// Mitsubishi GX Works2 project: BookEX6_10 String   PLC: Q13UDV

// global labels: Global
VAR_GLOBAL
  bVar0 AT M5000 : BOOL;
  abArray0 AT M5010 : ARRAY [0..49] OF BOOL;
  sStr0 AT D5000 : STRING[199];
  sStr1 AT D5100 : STRING[199];
  sStr2 AT D5200 : STRING[199];
  sStr3 AT D5300 : STRING[199];
  sStr4 AT D5400 : STRING[199];
  sStr5 AT D5500 : STRING[199];
  sStr6 AT D5600 : STRING[199];
  sStr7 AT D5700 : STRING[199];
  sStr8 AT D5800 : STRING[199];
  sStr9 AT D5900 : STRING[199];
  iVar0 AT D4500 : INT;
  iVar1 AT D4501 : INT;
  iVar2 AT D4502 : INT;
  iVar3 AT D4503 : INT;
  iVar4 AT D4504 : INT;
  iVar5 AT D4505 : INT;
  iVar6 AT D4506 : INT;
  iVar7 AT D4507 : INT;
  iVar8 AT D4508 : INT;
  iVar9 AT D4509 : INT;
  dVar0 AT D4510 : DINT;
  dVar1 AT D4512 : DINT;
  dVar2 AT D4514 : DINT;
  dVar3 AT D4516 : DINT;
  dVar4 AT D4518 : DINT;
  dVar5 AT D4520 : DINT;
  dVar6 AT D4522 : DINT;
  dVar7 AT D4524 : DINT;
  dVar8 AT D4526 : DINT;
  dVar9 AT D4528 : DINT;
  wVar0 AT D4530 : WORD;
  wVar1 AT D4531 : WORD;
  wVar2 AT D4532 : WORD;
  wVar3 AT D4533 : WORD;
  wVar4 AT D4534 : WORD;
  wVar5 AT D4535 : WORD;
  wVar6 AT D4536 : WORD;
  wVar7 AT D4537 : WORD;
  wVar8 AT D4538 : WORD;
  wVar9 AT D4539 : WORD;
  dwVar0 AT D4540 : DWORD;
  dwVar1 AT D4542 : DWORD;
  dwVar2 AT D4544 : DWORD;
  dwVar3 AT D4546 : DWORD;
  dwVar4 AT D4548 : DWORD;
  dwVar5 AT D4550 : DWORD;
  dwVar6 AT D4552 : DWORD;
  dwVar7 AT D4554 : DWORD;
  dwVar8 AT D4556 : DWORD;
  dwVar9 AT D4558 : DWORD;
  fsVar0 AT D4560 : REAL;
  fsVar1 AT D4562 : REAL;
  fsVar2 AT D4564 : REAL;
  fsVar3 AT D4566 : REAL;
  fsVar4 AT D4568 : REAL;
  fsVar5 AT D4570 : REAL;
  fsVar6 AT D4572 : REAL;
  fsVar7 AT D4574 : REAL;
  fsVar8 AT D4576 : REAL;
  fsVar9 AT D4578 : REAL;
  fdVar0 AT D4580 : LREAL;
  tTime0 AT D4620 : TIME;
  tTime1 AT D4622 : TIME;
  tTime2 AT D4624 : TIME;
  tTime3 AT D4626 : TIME;
  tTime4 AT D4628 : TIME;
  tTime5 AT D4630 : TIME;
  tTime6 AT D4632 : TIME;
  tTime7 AT D4634 : TIME;
  tTime8 AT D4636 : TIME;
  tTime9 AT D4638 : TIME;
  tTime10 AT D4640 : TIME;
  bVar1 AT M5001 : BOOL;
  bVar2 AT M5002 : BOOL;
  bVar3 AT M5003 : BOOL;
  bVar4 AT M5004 : BOOL;
  bVar5 AT M5005 : BOOL;
  bVar6 AT M5006 : BOOL;
  bVar7 AT M5007 : BOOL;
  bVar8 AT M5008 : BOOL;
  bVar9 AT M5009 : BOOL;
  abArray1 AT M5060 : ARRAY [0..49] OF BOOL;
  abArray2 AT M5110 : ARRAY [0..49] OF BOOL;
  abArray3 AT M5160 : ARRAY [0..49] OF BOOL;
  abArray4 AT M5210 : ARRAY [0..49] OF BOOL;
  abArray5 AT M5260 : ARRAY [0..49] OF BOOL;
  abArray6 AT M5310 : ARRAY [0..49] OF BOOL;
  abArray7 AT M5360 : ARRAY [0..49] OF BOOL;
  abArray8 AT M5410 : ARRAY [0..49] OF BOOL;
  abArray9 AT M5460 : ARRAY [0..49] OF BOOL;
  fdVar1 AT D4584 : LREAL;
  fdVar2 AT D4588 : LREAL;
  fdVar3 AT D4592 : LREAL;
  fdVar4 AT D4596 : LREAL;
  fdVar5 AT D4600 : LREAL;
  fdVar6 AT D4604 : LREAL;
  fdVar7 AT D4608 : LREAL;
  fdVar8 AT D4612 : LREAL;
  fdVar9 AT D4616 : LREAL;
END_VAR
// user libraries (not included): HMI

FUNCTION ChkALNUM
VAR_INPUT
  s_IN : STRING[199];
END_VAR
VAR
  ix : INT;
  iLeng : INT;
  iChar : INT;
  sTmpStr : STRING[199];
END_VAR
;
sTmpStr := s_IN;
LEN_E(TRUE, s_IN, iLeng);
IF iLeng = 0 THEN
	ChkALNUM := FALSE;
	RETURN;
END_IF;
FOR ix := 1 TO iLeng DO
	iChar := GET_INT_ADDR(sTmpStr) MOD 256;
	IF NOT ((iChar > H2F AND iChar < H3A) OR (iChar > H40 AND iChar < H5B) OR (iChar > H60 AND iChar < H7B)) THEN
		ChkALNUM := FALSE;
		RETURN;
	END_IF;
	sTmpStr := DELETE(sTmpStr, 1, 1);
END_FOR;
ChkALNUM := TRUE;
END_FUNCTION

FUNCTION ChkALPHA
VAR_INPUT
  s_IN : STRING[199];
END_VAR
VAR
  ix : INT;
  iLeng : INT;
  iChar : INT;
  sTmpStr : STRING[199];
END_VAR
;
sTmpStr := s_IN;
LEN_E(TRUE, s_IN, iLeng);
IF iLeng = 0 THEN
	ChkALPHA := FALSE;
	RETURN;
END_IF;
FOR ix := 1 TO iLeng DO
	iChar := GET_INT_ADDR(sTmpStr) MOD 256;
	IF NOT ((iChar > H40 AND iChar < H5B) OR (iChar > H60 AND iChar < H7B)) THEN
		ChkALPHA := FALSE;
		RETURN;
	END_IF;
	sTmpStr := DELETE(sTmpStr, 1, 1);
END_FOR;
ChkALPHA := TRUE;
END_FUNCTION

FUNCTION ChkHEXSTR
VAR_INPUT
  s_IN : STRING[199];
END_VAR
VAR
  ix : INT;
  iLeng : INT;
  iChar : INT;
  sTmpStr : STRING[199];
END_VAR
;
sTmpStr := s_IN;
LEN_E(TRUE, s_IN, iLeng);
IF iLeng = 0 THEN
	ChkHEXSTR := FALSE;
	RETURN;
END_IF;
FOR ix := 1 TO iLeng DO
	iChar := GET_INT_ADDR(sTmpStr) MOD 256;
	IF NOT ((iChar > H2F AND iChar < H3A) OR (iChar > H40 AND iChar < H47) OR (iChar > H60 AND iChar < H67)) THEN
		ChkHEXSTR := FALSE;
		RETURN;
	END_IF;
	sTmpStr := DELETE(sTmpStr, 1, 1);
END_FOR;
ChkHEXSTR := TRUE;
END_FUNCTION

FUNCTION ChkNUM
VAR_INPUT
  s_IN : STRING[199];
END_VAR
VAR
  ix : INT;
  iLeng : INT;
  iChar : INT;
  sTmpStr : STRING[199];
END_VAR
;
sTmpStr := s_IN;
LEN_E(TRUE, s_IN, iLeng);
IF iLeng = 0 THEN
	ChkNUM := FALSE;
	RETURN;
END_IF;
FOR ix := 1 TO iLeng DO
	iChar := GET_INT_ADDR(sTmpStr) MOD 256;
	IF NOT (iChar > H2F AND iChar < H3A) THEN
		ChkNUM := FALSE;
		RETURN;
	END_IF;
	sTmpStr := DELETE(sTmpStr, 1, 1);
END_FOR;
ChkNUM := TRUE;
END_FUNCTION

FUNCTION FindNUM
VAR_INPUT
  s_IN : STRING[199];
END_VAR
VAR
  ix : INT;
  iLeng : INT;
  iChar : INT;
  sTmpStr : STRING[199];
END_VAR
VAR_INPUT
  b_Num : BOOL;
END_VAR
;
sTmpStr := s_IN;
LEN_E(TRUE, s_IN, iLeng);
IF iLeng = 0 THEN
	FindNUM := 0;
	RETURN;
END_IF;
FOR ix := 1 TO iLeng DO
	iChar := GET_INT_ADDR(sTmpStr) MOD 256;
	IF (b_Num AND (iChar > H2F AND iChar < H3A)) OR 
		(NOT b_Num AND  NOT (iChar > H2F AND iChar < H3A)) THEN
		FindNUM := ix;
		RETURN;
	END_IF;
	sTmpStr := DELETE(sTmpStr, 1, 1);
END_FOR;
FindNUM := 0;
END_FUNCTION

FUNCTION MirrorStr
VAR_INPUT
  s_IN : STRING[199];
END_VAR
VAR
  ix : INT;
  iLeng : INT;
  sChar : STRING[1];
  sTmpStr : STRING[199];
  sTmpStr2 : STRING[199];
  sTmpStr1 : STRING[199];
END_VAR
;
sTmpStr := s_IN;
LEN_E(TRUE, s_IN, iLeng);
IF iLeng < 2 THEN
	MirrorStr := sTmpStr;
	RETURN;
END_IF;
sTmpStr2 := '';
FOR ix := iLeng TO 1 BY -1 DO 
	RIGHT_E(TRUE, sTmpStr, 1, sChar);
(*	STRDEL(TRUE, ix, 1, sTmpStr); *)
	sTmpStr1 := DELETE(sTmpStr, 1, ix);
	sTmpStr := sTmpStr1;
	sTmpStr2 := CONCAT(sTmpStr2, sChar);
END_FOR;  
MirrorStr := sTmpStr2;
END_FUNCTION

FUNCTION_BLOCK OperatingTime
VAR_INPUT
  b_Working : BOOL;  (* 설비의 작동상태 *)
END_VAR
VAR_OUTPUT
  d_WorkSec : DINT;  (* 경과 시간을 초로 표시 *)
  s_WorkStr : STRING[32];  (* 경과 시간을 문자열로 표시 *)
END_VAR
VAR
  TON_1 : TON;
  dWorkTime : DINT;
END_VAR
VAR_OUTPUT
  b_Work : BOOL;  (* 동작 램프 *)
  b_Warn : BOOL;  (* 경고 램프 *)
END_VAR
VAR
  dWorkDay : DINT;
  aiWorkHMS : ARRAY [0..2] OF INT;
  sWork : STRING[32];
  sTemp1 : STRING[32];
END_VAR
VAR_INPUT
  b_Clear : BOOL;  (* 동작시간 초기화 *)
  d_Day : DINT;  (* 경고시간중 일 *)
  d_Hour : DINT;  (* 경고시간중 시 *)
  d_Min : DINT;  (* 경고시간중 분 *)
  d_Sec : DINT;  (* 경고시간중 초 *)
END_VAR
VAR
  dWarnTime : DINT;
  sForm : DINT;
END_VAR
;
IF LDP(TRUE, b_Clear) THEN			
	dWorkTime := 0;
END_IF;

b_Work := b_Working;
IF b_Working THEN
	TON_1(IN:= b_Working, PT:= T#1s);
	IF TON_1.Q THEN
		dWarnTime := d_Day*86400+d_Hour*3600+d_Min*60+d_Sec;
		TON_1(IN:= FALSE);
		dWorkTime := dWorkTime + 1;				
		dWorkDay := dWorkTime / 86400;		
		HOUR(TRUE, dWorkTime MOD 86400, aiWorkHMS);	
		sForm := 3;
		DSTR(TRUE, sForm, dWorkDay, sTemp1);  
		sTemp1 := DELETE(sTemp1, 1, 1);						
		sWork := CONCAT( sTemp1, "일 ");  
		STR(TRUE, sForm, aiWorkHMS[0], sTemp1);
		sTemp1 := DELETE(sTemp1, 1, 1);
		sWork := CONCAT(sWork, sTemp1, "시 "); 
		STR(TRUE, sForm, aiWorkHMS[1], sTemp1);
		sTemp1 := DELETE(sTemp1, 1, 1);
		sWork := CONCAT(sWork, sTemp1, "분 "); 
		STR(TRUE, sForm, aiWorkHMS[2], sTemp1);
		sTemp1 := DELETE(sTemp1, 1, 1);
		sWork := CONCAT(sWork, sTemp1, "초"); 	
		d_WorkSec := dWorkTime;
		s_WorkStr := sWork; 
	END_IF;	
ELSE
 		s_WorkStr := "작동중지";
END_IF;

IF (dWorkTime > dWarnTime) AND (dWarnTime <> 0) THEN 
	b_Warn := SM412;
ELSE
	b_Warn := FALSE;
END_IF;
END_FUNCTION_BLOCK

FUNCTION_BLOCK SpinStr
VAR_INPUT
  bEN : BOOL;
  s_IN : STRING[199];
END_VAR
VAR
  iLeng : INT;
  sTmpStr : STRING[199];
  sChar : STRING[1];
END_VAR
VAR_OUTPUT
  bENO : BOOL;
  s_OUT : STRING[199];
END_VAR
VAR
  fbTimer : TON;
END_VAR
;
bENO := bEN;
IF LDP(TRUE, bEN) THEN
	sTmpStr := s_IN;
	LEN_E(TRUE, s_IN, iLeng);
END_IF;
IF NOT bEN OR iLeng = 0 THEN
	RETURN;
END_IF;

fbTimer(IN := TRUE , PT := T#1s);
IF NOT fbTimer.Q THEN
	RETURN;
END_IF;
fbTimer(IN := FALSE);
LEFT_E(TRUE, sTmpStr,1, sChar);
sTmpStr := DELETE(sTmpStr, 1, 1);
sTmpStr := CONCAT(sTmpStr,sChar);
s_OUT := sTmpStr;
END_FUNCTION_BLOCK

FUNCTION TrimStr
VAR_INPUT
  s_IN : STRING[199];
END_VAR
VAR
  ix : INT;
  iLeng : INT;
  iChar : INT;
  sTmpStr : STRING[199];
  sTmpStr1 : STRING[199];
END_VAR
;
sTmpStr := s_IN;
LEN_E(TRUE, s_IN, iLeng);
IF iLeng = 0 THEN
	RETURN;
END_IF;
 
REPEAT 
	ix := FIND(sTmpStr, ' ');
	IF ix > 0 THEN
(*	STRDEL(TRUE, ix, 1, sTmpStr); *)
	sTmpStr1 := DELETE(sTmpStr, 1, ix);
	sTmpStr := sTmpStr1;
	END_IF;
UNTIL ix = 0
END_REPEAT;  
TrimStr := sTmpStr;
END_FUNCTION

PROGRAM ExChkChar
VAR
  SpinStr_1 : SpinStr;
  sTmp1 : STRING[199];
  sTmp2 : STRING[199];
  sTmp3 : STRING[199];
  sTmp4 : STRING[199];
  sTmp5 : STRING[199];
END_VAR
(* structured ladder/FBD written out as ST: instructions are called as NAME(EN, inputs, outputs); _pN, _eN, _tN stand for wires *)
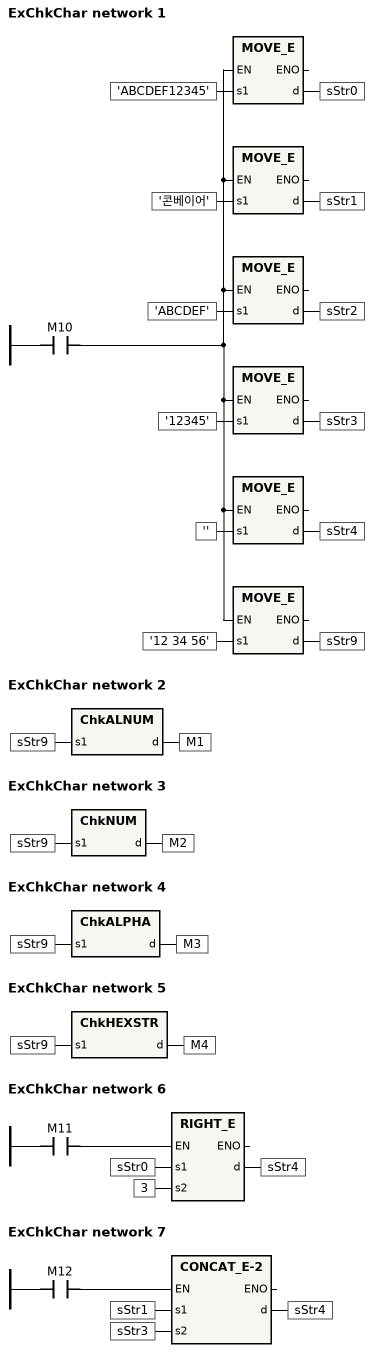
(* network 1 *)
MOVE_E(M10, 'ABCDEF12345', sStr0);
MOVE_E(M10, '콘베이어', sStr1);
MOVE_E(M10, 'ABCDEF', sStr2);
MOVE_E(M10, '12345', sStr3);
MOVE_E(M10, '', sStr4);
MOVE_E(M10, '12 34 56', sStr9);
(* network 2 *)
M1 := ChkALNUM(sStr9);
(* network 3 *)
M2 := ChkNUM(sStr9);
(* network 4 *)
M3 := ChkALPHA(sStr9);
(* network 5 *)
M4 := ChkHEXSTR(sStr9);
(* network 6 *)
RIGHT_E(M11, sStr0, 3, sStr4);
(* network 7 *)
CONCAT_E(M12, sStr1, sStr3, sStr4);
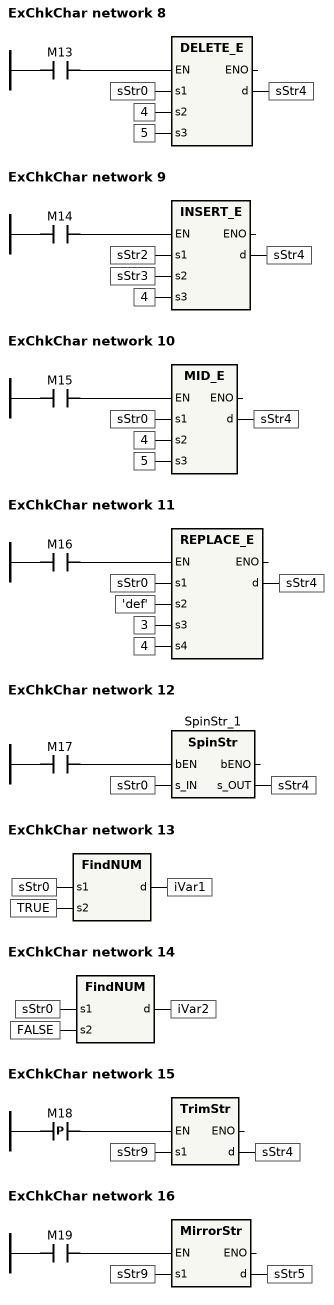
(* network 8 *)
DELETE_E(M13, sStr0, 4, 5, sStr4);
(* network 9 *)
INSERT_E(M14, sStr2, sStr3, 4, sStr4);
(* network 10 *)
MID_E(M15, sStr0, 4, 5, sStr4);
(* network 11 *)
REPLACE_E(M16, sStr0, 'def', 3, 4, sStr4);
(* network 12 *)
SpinStr_1(bEN := M17, s_IN := sStr0, s_OUT => sStr4);
(* network 13 *)
iVar1 := FindNUM(sStr0, TRUE);
(* network 14 *)
iVar2 := FindNUM(sStr0, FALSE);
(* network 15 *)
TrimStr(LDP(TRUE, M18), sStr9, sStr4);
(* network 16 *)
MirrorStr(M19, sStr9, sStr5);
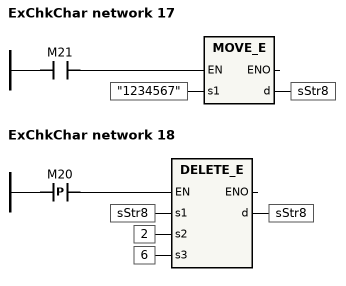
(* network 17 *)
MOVE_E(M21, "1234567", sStr8);
(* network 18 *)
DELETE_E(LDP(TRUE, M20), sStr8, 2, 6, sStr8);
END_PROGRAM

PROGRAM EXOpTime
VAR
  OperatingTime_1 : OperatingTime;
END_VAR
(* structured ladder/FBD written out as ST: instructions are called as NAME(EN, inputs, outputs); _pN, _eN, _tN stand for wires *)
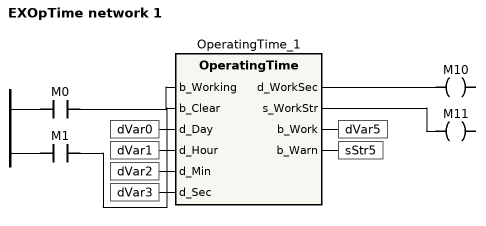
(* network 1 *)
OperatingTime_1(b_Working := M0, b_Clear := M1, d_Day := dVar0, d_Hour := dVar1, d_Min := dVar2, d_Sec := dVar3, b_Work => dVar5, b_Warn => sStr5);
M10 := OperatingTime_1.d_WorkSec;
M11 := OperatingTime_1.s_WorkStr;
END_PROGRAM

PROGRAM ExString
VAR
  Var_D0 : WORD;
  Var_D1 : INT;
  CTD_E_1 : CTD_E;
  COUNTER_FB_M_1 : COUNTER_FB_M;
  aiNo : ARRAY [0..5] OF INT;
  aiSno : ARRAY [0..1] OF INT;
  sTmpStr1 : STRING[199];
  sTmpStr2 : STRING[199];
  sTmpStr3 : STRING[199];
  sTmpStr4 : STRING[199];
  sTmpStr5 : STRING[199];
  sTmpStr6 : STRING[199];
  sTmpStr7 : STRING[199];
  sTmpStr8 : STRING[199];
  sTmpStr9 : STRING[199];
END_VAR
(* structured ladder/FBD written out as ST: instructions are called as NAME(EN, inputs, outputs); _pN, _eN, _tN stand for wires *)
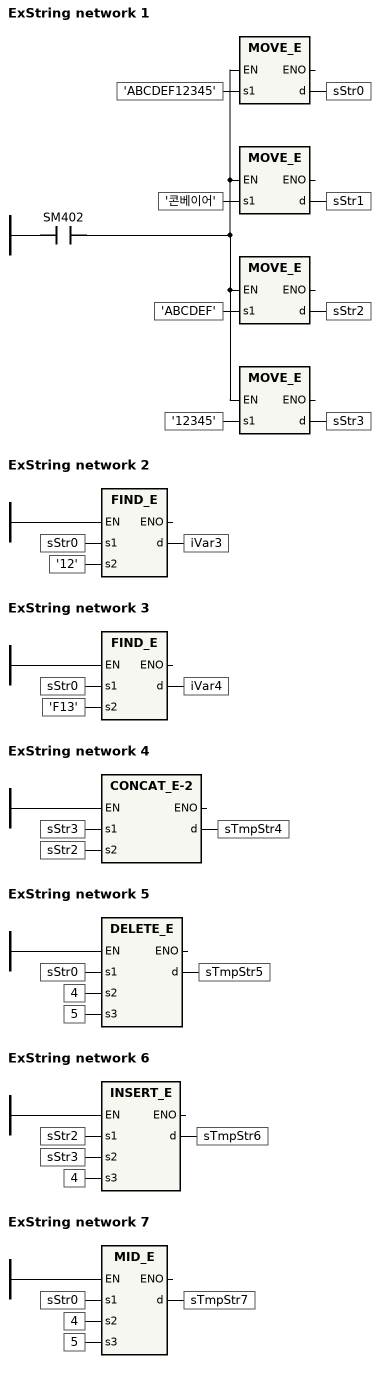
(* network 1 *)
MOVE_E(SM402, 'ABCDEF12345', sStr0);
MOVE_E(SM402, '콘베이어', sStr1);
MOVE_E(SM402, 'ABCDEF', sStr2);
MOVE_E(SM402, '12345', sStr3);
(* network 2 *)
FIND_E(TRUE, sStr0, '12', iVar3);
(* network 3 *)
FIND_E(TRUE, sStr0, 'F13', iVar4);
(* network 4 *)
CONCAT_E(TRUE, sStr3, sStr2, sTmpStr4);
(* network 5 *)
DELETE_E(TRUE, sStr0, 4, 5, sTmpStr5);
(* network 6 *)
INSERT_E(TRUE, sStr2, sStr3, 4, sTmpStr6);
(* network 7 *)
MID_E(TRUE, sStr0, 4, 5, sTmpStr7);
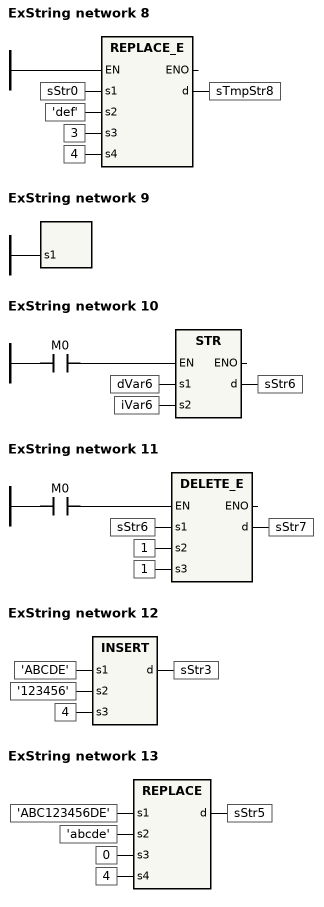
(* network 8 *)
REPLACE_E(TRUE, sStr0, 'def', 3, 4, sTmpStr8);
(* network 9 *)
(* element kind 10  <- TRUE *)
(* network 10 *)
STR(M0, dVar6, iVar6, sStr6);
(* network 11 *)
DELETE_E(M0, sStr6, 1, 1, sStr7);
(* network 12 *)
sStr3 := INSERT('ABCDE', '123456', 4);
(* network 13 *)
sStr5 := REPLACE('ABC123456DE', 'abcde', 0, 4);
END_PROGRAM

PROGRAM ExLEN
VAR
  Var_D0 : WORD;
  Var_D1 : INT;
  CTD_E_1 : CTD_E;
  COUNTER_FB_M_1 : COUNTER_FB_M;
  aiNo : ARRAY [0..5] OF INT;
  aiSno : ARRAY [0..1] OF INT;
  sTmpStr1 : STRING[199];
  sTmpStr2 : STRING[199];
  sTmpStr3 : STRING[199];
  sTmpStr4 : STRING[199];
  sTmpStr5 : STRING[199];
  sTmpStr6 : STRING[199];
  sTmpStr7 : STRING[199];
  sTmpStr8 : STRING[199];
  sTmpStr9 : STRING[199];
END_VAR
(* structured ladder/FBD written out as ST: instructions are called as NAME(EN, inputs, outputs); _pN, _eN, _tN stand for wires *)
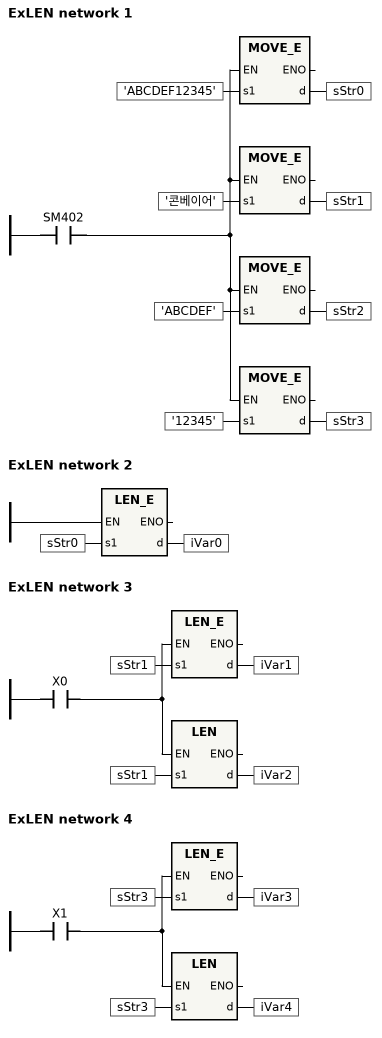
(* network 1 *)
MOVE_E(SM402, 'ABCDEF12345', sStr0);
MOVE_E(SM402, '콘베이어', sStr1);
MOVE_E(SM402, 'ABCDEF', sStr2);
MOVE_E(SM402, '12345', sStr3);
(* network 2 *)
LEN_E(TRUE, sStr0, iVar0);
(* network 3 *)
LEN_E(X0, sStr1, iVar1);
LEN(X0, sStr1, iVar2);
(* network 4 *)
LEN_E(X1, sStr3, iVar3);
LEN(X1, sStr3, iVar4);
END_PROGRAM

PROGRAM ExLEFT
VAR
  Var_D0 : WORD;
  Var_D1 : INT;
  CTD_E_1 : CTD_E;
  COUNTER_FB_M_1 : COUNTER_FB_M;
  aiNo : ARRAY [0..5] OF INT;
  aiSno : ARRAY [0..1] OF INT;
  sTmpStr1 : STRING[199];
  sTmpStr2 : STRING[199];
  sTmpStr3 : STRING[199];
  sTmpStr4 : STRING[199];
  sTmpStr5 : STRING[199];
  sTmpStr6 : STRING[199];
  sTmpStr7 : STRING[199];
  sTmpStr8 : STRING[199];
  sTmpStr9 : STRING[199];
END_VAR
(* structured ladder/FBD written out as ST: instructions are called as NAME(EN, inputs, outputs); _pN, _eN, _tN stand for wires *)
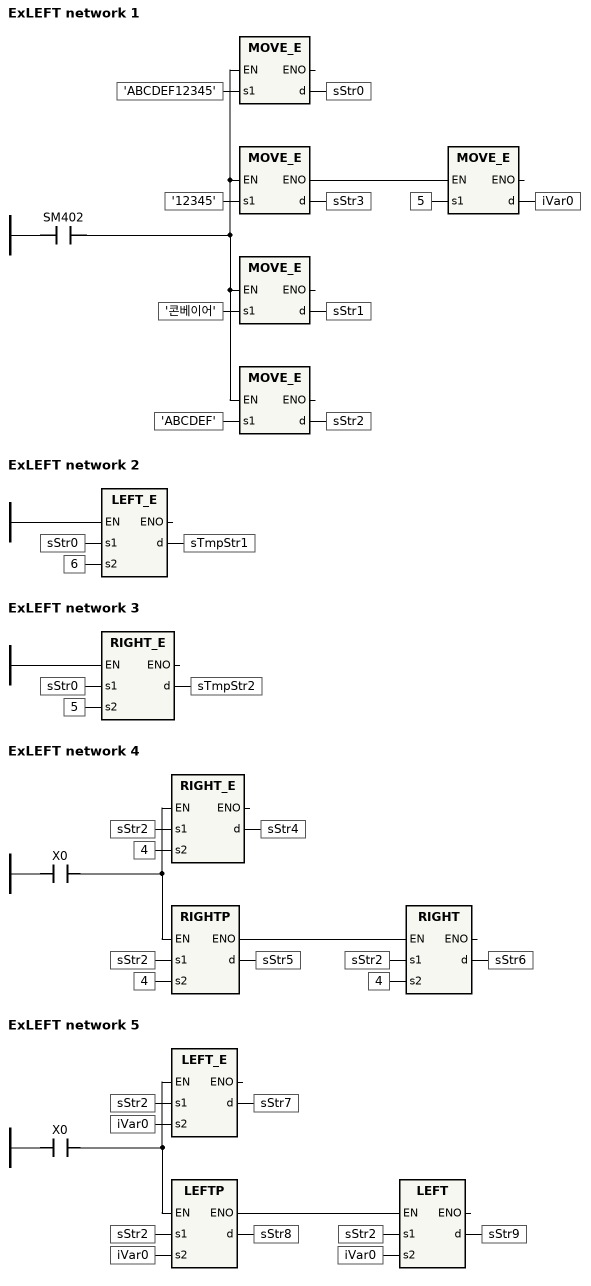
(* network 1 *)
MOVE_E(SM402, 'ABCDEF12345', sStr0);
MOVE_E(SM402, '콘베이어', sStr1);
MOVE_E(SM402, 'ABCDEF', sStr2);
_e1 := MOVE_E(SM402, '12345', sStr3);
MOVE_E(_e1, 5, iVar0);
(* network 2 *)
LEFT_E(TRUE, sStr0, 6, sTmpStr1);
(* network 3 *)
RIGHT_E(TRUE, sStr0, 5, sTmpStr2);
(* network 4 *)
RIGHT_E(X0, sStr2, 4, sStr4);
_e1 := RIGHTP(X0, sStr2, 4, sStr5);
RIGHT(_e1, sStr2, 4, sStr6);
(* network 5 *)
LEFT_E(X0, sStr2, iVar0, sStr7);
_e1 := LEFTP(X0, sStr2, iVar0, sStr8);
LEFT(_e1, sStr2, iVar0, sStr9);
END_PROGRAM

PROGRAM ExCONCAT
VAR
  Var_D0 : WORD;
  Var_D1 : INT;
  CTD_E_1 : CTD_E;
  COUNTER_FB_M_1 : COUNTER_FB_M;
  aiNo : ARRAY [0..5] OF INT;
  aiSno : ARRAY [0..1] OF INT;
  sTmpStr1 : STRING[199];
  sTmpStr2 : STRING[199];
  sTmpStr3 : STRING[199];
  sTmpStr4 : STRING[199];
  sTmpStr5 : STRING[199];
  sTmpStr6 : STRING[199];
  sTmpStr7 : STRING[199];
  sTmpStr8 : STRING[199];
  sTmpStr9 : STRING[199];
END_VAR
(* structured ladder/FBD written out as ST: instructions are called as NAME(EN, inputs, outputs); _pN, _eN, _tN stand for wires *)
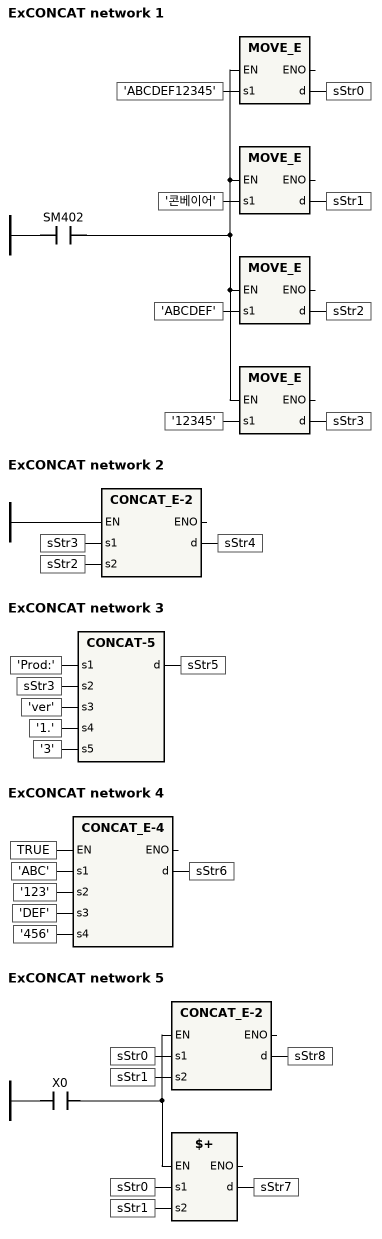
(* network 1 *)
MOVE_E(SM402, 'ABCDEF12345', sStr0);
MOVE_E(SM402, '콘베이어', sStr1);
MOVE_E(SM402, 'ABCDEF', sStr2);
MOVE_E(SM402, '12345', sStr3);
(* network 2 *)
CONCAT_E(TRUE, sStr3, sStr2, sStr4);
(* network 3 *)
sStr5 := CONCAT('Prod:', sStr3, 'ver', '1.', '3');
(* network 4 *)
CONCAT_E(TRUE, 'ABC', '123', 'DEF', '456', sStr6);
(* network 5 *)
CONCAT_E(X0, sStr0, sStr1, sStr8);
$+(X0, sStr0, sStr1, sStr7);
END_PROGRAM

PROGRAM ExDELETE
VAR
  Var_D0 : WORD;
  Var_D1 : INT;
  CTD_E_1 : CTD_E;
  COUNTER_FB_M_1 : COUNTER_FB_M;
  aiNo : ARRAY [0..5] OF INT;
  aiSno : ARRAY [0..1] OF INT;
  sTmpStr1 : STRING[199];
  sTmpStr2 : STRING[199];
  sTmpStr3 : STRING[199];
  sTmpStr4 : STRING[199];
  sTmpStr5 : STRING[199];
  sTmpStr6 : STRING[199];
  sTmpStr7 : STRING[199];
  sTmpStr8 : STRING[199];
  sTmpStr9 : STRING[199];
END_VAR
(* structured ladder/FBD written out as ST: instructions are called as NAME(EN, inputs, outputs); _pN, _eN, _tN stand for wires *)
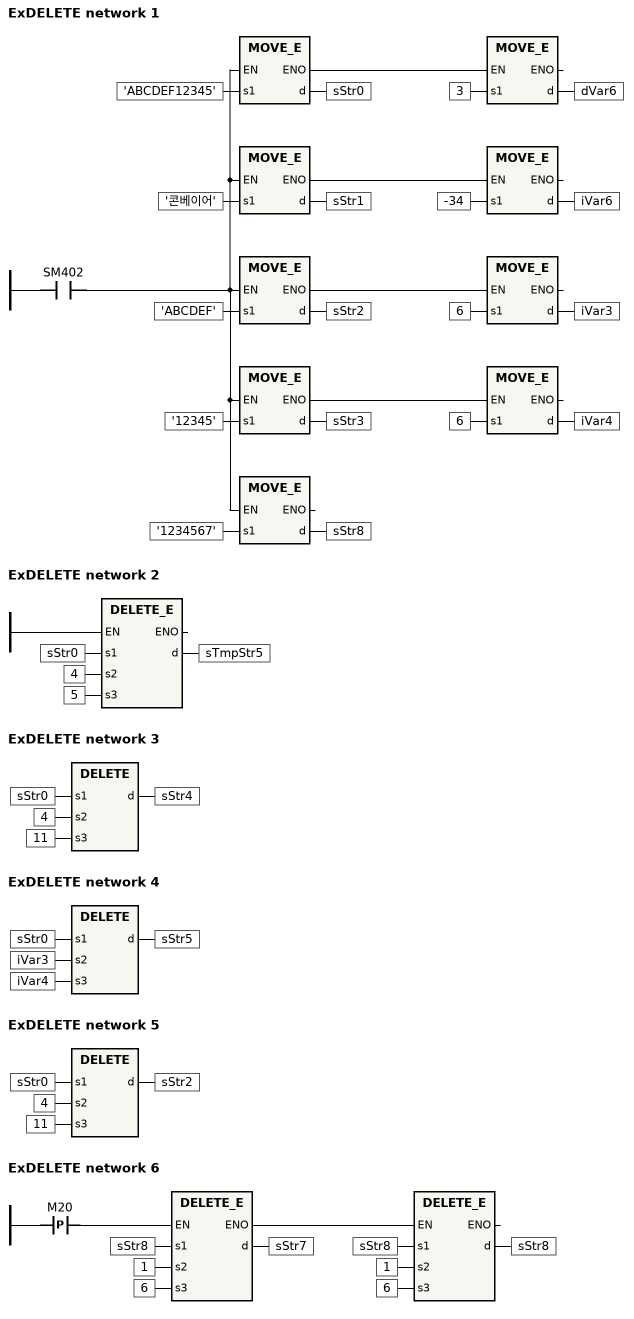
(* network 1 *)
_e1 := MOVE_E(SM402, 'ABCDEF12345', sStr0);
MOVE_E(_e1, 3, dVar6);
_e2 := MOVE_E(SM402, '콘베이어', sStr1);
MOVE_E(_e2, -34, iVar6);
_e3 := MOVE_E(SM402, 'ABCDEF', sStr2);
MOVE_E(_e3, 6, iVar3);
_e4 := MOVE_E(SM402, '12345', sStr3);
MOVE_E(_e4, 6, iVar4);
MOVE_E(SM402, '1234567', sStr8);
(* network 2 *)
DELETE_E(TRUE, sStr0, 4, 5, sTmpStr5);
(* network 3 *)
sStr4 := DELETE(sStr0, 4, 11);
(* network 4 *)
sStr5 := DELETE(sStr0, iVar3, iVar4);
(* network 5 *)
sStr2 := DELETE(sStr0, 4, 11);
(* network 6 *)
_e1 := DELETE_E(LDP(TRUE, M20), sStr8, 1, 6, sStr7);
DELETE_E(_e1, sStr8, 1, 6, sStr8);
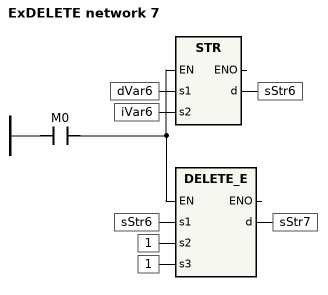
(* network 7 *)
STR(M0, dVar6, iVar6, sStr6);
DELETE_E(M0, sStr6, 1, 1, sStr7);
END_PROGRAM

PROGRAM ExMID
VAR
  Var_D0 : WORD;
  Var_D1 : INT;
  CTD_E_1 : CTD_E;
  COUNTER_FB_M_1 : COUNTER_FB_M;
  aiNo : ARRAY [0..5] OF INT;
  aiSno : ARRAY [0..1] OF INT;
  sTmpStr1 : STRING[199];
  sTmpStr2 : STRING[199];
  sTmpStr3 : STRING[199];
  sTmpStr4 : STRING[199];
  sTmpStr5 : STRING[199];
  sTmpStr6 : STRING[199];
  sTmpStr7 : STRING[199];
  sTmpStr8 : STRING[199];
  sTmpStr9 : STRING[199];
  aiVar0 : ARRAY [0..1] OF INT;
  aiVar1 : ARRAY [0..1] OF INT;
END_VAR
(* structured ladder/FBD written out as ST: instructions are called as NAME(EN, inputs, outputs); _pN, _eN, _tN stand for wires *)
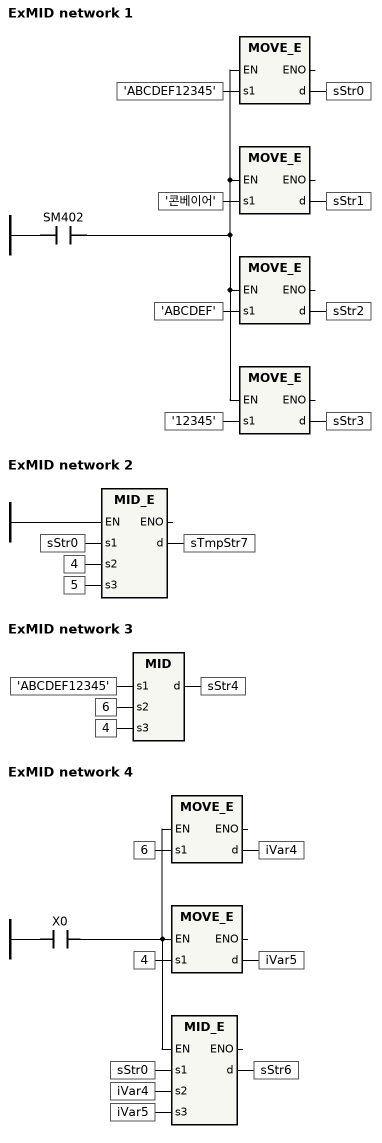
(* network 1 *)
MOVE_E(SM402, 'ABCDEF12345', sStr0);
MOVE_E(SM402, '콘베이어', sStr1);
MOVE_E(SM402, 'ABCDEF', sStr2);
MOVE_E(SM402, '12345', sStr3);
(* network 2 *)
MID_E(TRUE, sStr0, 4, 5, sTmpStr7);
(* network 3 *)
sStr4 := MID('ABCDEF12345', 6, 4);
(* network 4 *)
MOVE_E(X0, 6, iVar4);
MOVE_E(X0, 4, iVar5);
MID_E(X0, sStr0, iVar4, iVar5, sStr6);
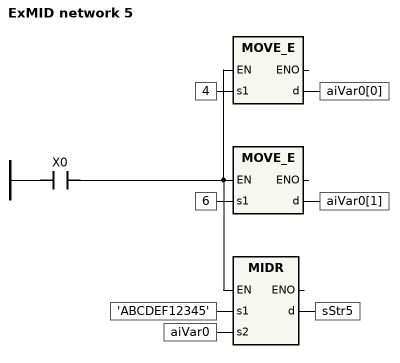
(* network 5 *)
MOVE_E(X0, 4, aiVar0[0]);
MOVE_E(X0, 6, aiVar0[1]);
MIDR(X0, 'ABCDEF12345', aiVar0, sStr5);
END_PROGRAM

PROGRAM ExLEN_ST
VAR
  iDataLen : INT;
  bNG : BOOL;
  bScanComp : BOOL;
END_VAR
;


IF bScanComp THEN				(*  스캔이 완료되었을 때 글자 수를 측정 *)
    LEN_E(TRUE, sStr0, iDataLen );
        
    IF iDataLen <> 8 THEN		(*. 바코드가 8자리인지 검사 *)
    	bNG := TRUE;  (* 불량 배출 실린더 ON *)
    ELSE
        bNG := FALSE; (* 정상 통과 *)
    END_IF;
    
    bScanComp := FALSE;    (* 완료 플래그 리셋*)
END_IF;
END_PROGRAM

PROGRAM ExLEFT_ST
VAR
  sScanData : STRING[32];
  sFactoryCode : STRING[32];
  sSerialNo : STRING[32];
END_VAR
;

sScanData := "ABC01-2026-123";			(* Test를 위한 데이터 *)
(* 맨 왼쪽에서 5글자를 추출*)
LEFT_E(TRUE, sScanData, 5, sFactoryCode );  	(* 결과: 'ABC01' *)

(* 오른쪽에서 3글자를 추출 *)
RIGHT(TRUE, sScanData, 3, sSerialNo );					(* 결과: '123' *)
iVar0 := STR_TO_INT(sSerialNo);					(* 결과: '23000' *)
iVar1 := newVAL(sSerialNo);					(* 결과:123 *)
END_PROGRAM

FUNCTION newVAL
VAR_INPUT
  s_IN : STRING[199];
END_VAR
VAR
  ix : INT;
  iChar : INT;
  iLeng : INT;
  sTmpStr : STRING[199];
  iVal : INT;
END_VAR
;
sTmpStr := s_IN;
LEN_E(TRUE, s_IN, iLeng);
IF iLeng = 0 THEN
	newVAL:= 0;
	RETURN;
END_IF;
iVal := 0;
FOR ix := 1 TO iLeng DO
	iChar := GET_INT_ADDR(sTmpStr) MOD 256;
	IF NOT (iChar > H2F AND iChar < H3A) THEN
		newVAL:= 0;
		RETURN;
	END_IF;
	iVal := (iChar - H30) + iVal * 10;
	sTmpStr := DELETE(sTmpStr, 1, 1);
END_FOR;
newVAL:= iVal;
END_FUNCTION

FUNCTION FILL
VAR_INPUT
  b_EN : BOOL;
  s_Str : STRING[32];
END_VAR
VAR
  ix : INT;
END_VAR
VAR_INPUT
  i_Len : INT;
END_VAR
VAR
  sTemp : STRING[199];
END_VAR
;
LEN(TRUE, s_Str, ix);
IF NOT b_EN OR (i_Len*ix) > 199 THEN
	FILL := '';
	RETURN;
END_IF;
sTemp := '';
FOR ix := 1 TO i_Len DO
	sTemp := CONCAT(sTemp,s_Str);
END_FOR;
FILL := sTemp;
END_FUNCTION

PROGRAM ExLeftRight
(* structured ladder/FBD written out as ST: instructions are called as NAME(EN, inputs, outputs); _pN, _eN, _tN stand for wires *)
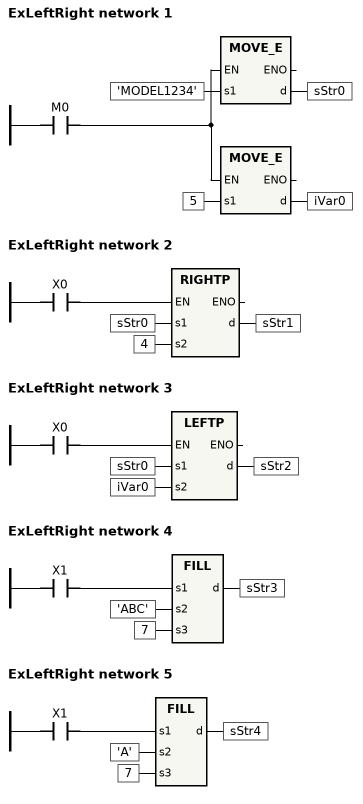
(* network 1 *)
MOVE_E(M0, 'MODEL1234', sStr0);
MOVE_E(M0, 5, iVar0);
(* network 2 *)
RIGHTP(X0, sStr0, 4, sStr1);
(* network 3 *)
LEFTP(X0, sStr0, iVar0, sStr2);
(* network 4 *)
sStr3 := FILL(X1, 'ABC', 7);
(* network 5 *)
sStr4 := FILL(X1, 'A', 7);
END_PROGRAM
